  def rq_current_pos_mm(gripper_socket=1):
      pos_gripper = rq_current_pos(gripper_socket)
      pos_mm = gripper_to_mm(pos_gripper, gripper_socket)
      return round_value_2_dec(pos_mm)
  end

  def rq_current_pos_inches(gripper_socket=1):
      pos_gripper = rq_current_pos(gripper_socket)
      pos_mm = gripper_to_mm(pos_gripper, gripper_socket)
      pos_in = pos_mm / 25.4
      return round_value_2_dec(pos_in)
  end

  def rq_move_mm(pos_mm, gripper_socket=1):
      pos_gripper = mm_to_gripper(pos_mm, gripper_socket)
      rq_move(pos_gripper, gripper_socket)
  end

  def rq_move_and_wait_mm(pos_mm, gripper_socket=1):
      pos_gripper = mm_to_gripper(pos_mm, gripper_socket)
      rq_move_and_wait(pos_gripper, gripper_socket)
  end

  def rq_move_inches(pos_in, gripper_socket=1):
      pos_mm = pos_in * 25.4
      rq_move_mm(pos_mm, gripper_socket)
  end

  def rq_move_and_wait_inches(pos_in, gripper_socket=1):
      pos_mm = pos_in * 25.4
      rq_move_and_wait_mm(pos_mm, gripper_socket)
  end

  def get_closed_norm(gripper_socket):
      return gripper_closed_norm[gripper_socket - 1]
  end

  def get_open_norm(gripper_socket):
      return gripper_open_norm[gripper_socket - 1]
  end

  def get_closed_mm(gripper_socket):
      return gripper_closed_mm[gripper_socket - 1]
  end

  def get_open_mm(gripper_socket):
      return gripper_open_mm[gripper_socket - 1]
  end

  def set_closed_norm(closed_norm, gripper_socket):
      gripper_closed_norm[gripper_socket - 1] = closed_norm
  end

  def set_open_norm(open_norm, gripper_socket):
      gripper_open_norm[gripper_socket - 1] = open_norm
  end

  def set_closed_mm(closed_mm, gripper_socket):
      gripper_closed_mm[gripper_socket - 1] = closed_mm
  end

  def set_open_mm(open_mm, gripper_socket):
      gripper_open_mm[gripper_socket - 1] = open_mm
  end

  def gripper_to_mm(value_gripper, gripper_socket):
      closed_norm = get_closed_norm(gripper_socket)
      open_norm = get_open_norm(gripper_socket)
      closed_mm = get_closed_mm(gripper_socket)
      open_mm = get_open_mm(gripper_socket)

      value_norm = (value_gripper / 255) * 100

      slope = (closed_mm - open_mm) / (closed_norm - open_norm)
      value_mm = slope * (value_norm - closed_norm) + closed_mm

      if (value_mm > open_mm):
          value_mm_limited = open_mm
      elif (value_mm < closed_mm):
          value_mm_limited = closed_mm
      else:
          value_mm_limited = value_mm
      end

      return value_mm_limited
  end

  def mm_to_gripper(value_mm, gripper_socket):
      closed_norm = get_closed_norm(gripper_socket)
      open_norm = get_open_norm(gripper_socket)
      closed_mm = get_closed_mm(gripper_socket)
      open_mm = get_open_mm(gripper_socket)

      slope = (closed_norm - open_norm) / (closed_mm - open_mm)
      value_norm = (value_mm - closed_mm) * slope + closed_norm

      value_gripper = value_norm * 255 / 100

      if (value_gripper > 255):
          value_gripper_limited = 255
      elif (value_gripper < 0):
          value_gripper_limited = 0
      else:
          value_gripper_limited = round_value(value_gripper)
      end

      return value_gripper_limited
  end

  def round_value(value):
      value_mod = value % 1

      if(value_mod < 0.5):
          return floor(value)
      else:
          return ceil(value)
      end
  end

  def round_value_2_dec(value):
      value_x_100 = value * 100
      value_x_100_rounded = round_value(value_x_100)
      return value_x_100_rounded / 100
  end

  def clear_socket_buffer(gripper_socket="1", read_timeout = 0.1):
    byte_in_buffer = socket_read_byte_list(1, gripper_socket, read_timeout)

    while(byte_in_buffer[0] >= 1):
        byte_in_buffer = socket_read_byte_list(1, gripper_socket, read_timeout)
    end
  end

  def rq_set_gripper_socket_acquire_option(enabled=False):
      gripper_socket_acquire_option = enabled

      if(not enabled):
          gripper_1_socket_acquired = False
          gripper_2_socket_acquired = False
          gripper_3_socket_acquired = False
          gripper_4_socket_acquired = False
      end
  end

  def rq_acquire_gripper_socket(gripper_socket="1"):
      if(gripper_socket_acquire_option):
          rq_wait_gripper_socket_released(gripper_socket)
          enter_critical
              rq_set_gripper_socket_acquired(gripper_socket, True)
          exit_critical

          clear_socket_buffer(gripper_socket, 0.002)

          sync()
      end
  end

  def rq_release_gripper_socket(gripper_socket="1"):
      if(gripper_socket_acquire_option):
          rq_set_gripper_socket_acquired(gripper_socket, False)

          sync()
      end
  end

  def rq_set_gripper_socket_acquired(gripper_socket="1", acquired=False):
      if(gripper_socket == "1"):
          gripper_1_socket_acquired = acquired
      elif(gripper_socket == "2"):
          gripper_2_socket_acquired = acquired
      elif(gripper_socket == "3"):
          gripper_3_socket_acquired = acquired
      elif(gripper_socket == "4"):
          gripper_4_socket_acquired = acquired
      end
  end

  def rq_get_gripper_socket_acquired(gripper_socket="1"):
      if(gripper_socket == "1"):
          return gripper_1_socket_acquired
      elif(gripper_socket == "2"):
          return gripper_2_socket_acquired
      elif(gripper_socket == "3"):
          return gripper_3_socket_acquired
      elif(gripper_socket == "4"):
          return gripper_4_socket_acquired
      end

      sync()
  end

  def rq_wait_gripper_socket_released(gripper_socket="1"):
      while(rq_get_gripper_socket_acquired(gripper_socket)):
          sync()
      end

      sync()
  end

  def scale(value, rawRange, scaledRange):
      def computeSlope(inputRange, outputRange):
          outputRangeDelta = outputRange[1] - outputRange[0]
          inputRangeDelta = inputRange[1] - inputRange[0]

          if (inputRangeDelta == 0):
              return 0
          else:
              return outputRangeDelta / inputRangeDelta
          end
      end

      def computeIntercept(slope, inputRange, outputRange):
          return outputRange[0] - (slope * inputRange[0])
      end

      def clipScaledValue(outputScaledValue, outputRange):
          if (outputRange[0] < outputRange[1]):
              return clipWhenLowerLimitIsLessThanHigher(outputScaledValue, outputRange)
          else:
              return clipWhenLowerLimitIsGreaterThanHigherLimit(outputScaledValue, outputRange)
          end
      end

      def clipWhenLowerLimitIsGreaterThanHigherLimit(outputScaledValue, outputRange):
          if (outputScaledValue < outputRange[1]):
              return outputRange[1]
          elif (outputScaledValue > outputRange[0]):
              return outputRange[0]
          else:
              return outputScaledValue
          end
      end

      def clipWhenLowerLimitIsLessThanHigher(outputScaledValue, outputRange):
          if (outputScaledValue < outputRange[0]):
              return outputRange[0]
          elif (outputScaledValue > outputRange[1]):
              return outputRange[1]
          else:
              return outputScaledValue
          end
      end

      slope = computeSlope(rawRange, scaledRange)
      intercept = computeIntercept(slope, rawRange, scaledRange)
      scaledValue = slope * value + intercept
      return clipScaledValue(scaledValue, scaledRange)
  end

  def limit(value, range):
      return scale(value, range, range)
  end


  rq_obj_detect = 0
  rq_init_comm_if_connected(9, "1")
  rq_init_comm_if_connected(2, "2")
  rq_init_comm_if_connected(3, "3")
  rq_init_comm_if_connected(4, "4")
  rq_print_connected_grippers()
  connectivity_checked = [-1,-1,-1,-1]
  status_checked = [-1,-1,-1,-1]
  current_speed = [-1,-1,-1,-1]
  current_force = [-1,-1,-1,-1]
  set_closed_norm(100.0, 1)
  set_open_norm(0.0, 1)
  set_closed_mm(0.0, 1)
  set_open_mm(50.0, 1)
  set_closed_norm(100.0, 2)
  set_open_norm(0.0, 2)
  set_closed_mm(0.0, 2)
  set_open_mm(50.0, 2)
  set_closed_norm(100.0, 3)
  set_open_norm(0.0, 3)
  set_closed_mm(0.0, 3)
  set_open_mm(50.0, 3)
  set_closed_norm(100.0, 4)
  set_open_norm(0.0, 4)
  set_closed_mm(0.0, 4)
  set_open_mm(50.0, 4)
  # end: URCap Installation Node
  $ 1 "BeforeStart"
  $ 2 "var_1≔ False "
  global var_1=  False
  $ 3 "thread_flag≔ False "
  global thread_flag=  False
  $ 4 "var_10≔[0,0,0,0,0,0,0,0,0,0]"
  global var_10=[0,0,0,0,0,0,0,0,0,0]
  $ 5 "Set"
  set_tcp(p[0.0,0.0,0.11,0.0,0.0,0.0])
  $ 198 "Thread_1"
  thread Thread_1():
    while (True):
      $ 199 "Loop thread_flag== False "
      while (thread_flag==  False  ):
        $ 200 "var_12=0"
        var_12=0
        $ 201 "Wait: 0.01"
        sleep(0.01)
      end
      $ 202 "Wait: 0.001"
      sleep(0.001)
      $ 203 "var_11≔get_tcp_force()"
      global var_11=get_tcp_force()
      $ 204 "If var_11[axis]*var_11[axis]<var_2[11]*var_2[11]"
      if (var_11[axis]*var_11[axis]<var_2[11]*var_2[11]):
        $ 205 "var_12=0"
        var_12=0
      else:
        $ 206 "Else"
        $ 207 "var_12=var_12+1"
        var_12=var_12+1
        $ 208 "If var_12>0"
        if (var_12>0):
          $ 209 "thread_flag= False "
          thread_flag=  False
        end
      end
    end
  end
  threadId_Thread_1 = run Thread_1()
  while (True):
    $ 6 "Robot Program"
    $ 7 "Loop var_1==False"
    while (var_1==False):
      $ 8 "var_1≔socket_open('192.168.1.5',30010)"
      global var_1=socket_open("192.168.1.5",30010)
      $ 9 "Wait: 0.5"
      sleep(0.5)
    end
    $ 10 "Loop var_1== True "
    thread Thread_while_10():
      while (True):
        $ 11 "Wait: 0.001"
        sleep(0.001)
        $ 12 "var_2≔socket_read_ascii_float(12)"
        global var_2=socket_read_ascii_float(12)
        $ 13 "Loop var_2[0]≠12"
        while (var_2[0] != 12):
          $ 14 "var_2≔socket_read_ascii_float(12)"
          global var_2=socket_read_ascii_float(12)
        end
        $ 15 "Switch var_2[1]"
        switch_1 = var_2[1]
        $ 16 "Case 0"
        if (0 == switch_1):
          $ 17 "'movejl'"
          # 'movejl'
          $ 18 "var_3≔p[var_2[2],var_2[3],var_2[4],var_2[5],var_2[6],var_2[7]]"
          global var_3=p[var_2[2],var_2[3],var_2[4],var_2[5],var_2[6],var_2[7]]
          $ 19 "movej(var_3,var_2[8],var_2[9],var_2[10],var_2[11])"
          movej(var_3,var_2[8],var_2[9],var_2[10],var_2[11])
          $ 20 "If var_2[12]==0"
          if (var_2[12]==0):
            $ 21 "socket_send_string('completed_pose_move')"
            socket_send_string("completed_pose_move")
          end
        elif (1 == switch_1):
          $ 22 "Case 1"
          $ 23 "'movej'"
          # 'movej'
          $ 24 "var_6≔[var_2[2],var_2[3],var_2[4],var_2[5],var_2[6],var_2[7]]"
          global var_6=[var_2[2],var_2[3],var_2[4],var_2[5],var_2[6],var_2[7]]
          $ 25 "movej(var_6,var_2[8],var_2[9],var_2[10],var_2[11])"
          movej(var_6,var_2[8],var_2[9],var_2[10],var_2[11])
          $ 26 "If var_2[12]==0"
          if (var_2[12]==0):
            $ 27 "socket_send_string('completed_joint_move')"
            socket_send_string("completed_joint_move")
          end
        elif (2 == switch_1):
          $ 28 "Case 2"
          $ 29 "'movel'"
          # 'movel'
          $ 30 "var_3≔p[var_2[2],var_2[3],var_2[4],var_2[5],var_2[6],var_2[7]]"
          global var_3=p[var_2[2],var_2[3],var_2[4],var_2[5],var_2[6],var_2[7]]
          $ 31 "movel(var_3,var_2[8],var_2[9],var_2[10],var_2[11])"
          movel(var_3,var_2[8],var_2[9],var_2[10],var_2[11])
          $ 32 "If var_2[12]==0"
          if (var_2[12]==0):
            $ 33 "socket_send_string('completed_linear_move')"
            socket_send_string("completed_linear_move")
          end
        elif (3 == switch_1):
          $ 34 "Case 3"
          $ 35 "'move to var_3 relative to current pose'"
          # 'move to var_3 relative to current pose'
          $ 36 "var_3≔p[var_2[2],var_2[3],var_2[4],var_2[5],var_2[6],var_2[7]]"
          global var_3=p[var_2[2],var_2[3],var_2[4],var_2[5],var_2[6],var_2[7]]
          $ 37 "var_5≔get_actual_tcp_pose()"
          global var_5=get_actual_tcp_pose()
          $ 38 "movel(pose_trans(var_5,var_3),var_2[8],var_2[9],var_2[10],var_2[11])"
          movel(pose_trans(var_5,var_3),var_2[8],var_2[9],var_2[10],var_2[11])
          $ 39 "If var_2[12]==0"
          if (var_2[12]==0):
            $ 40 "socket_send_string('completed_relative_linear_move')"
            socket_send_string("completed_relative_linear_move")
          end
        elif (4 == switch_1):
          $ 41 "Case 4"
          $ 42 "'force move in single axis'"
          # 'force move in single axis'
          $ 43 "var_5≔get_actual_tcp_pose()"
          global var_5=get_actual_tcp_pose()
          $ 44 "If var_2[2]≠0"
          if (var_2[2] != 0):
            $ 45 "var_5[0]=var_5[0]+var_2[2]"
            var_5[0]=var_5[0]+var_2[2]
            $ 46 "axis≔0"
            global axis=0
          else:
            $ 47 "ElseIf var_2[3]≠0"
            if (var_2[3] != 0):
              $ 48 "var_5[1]=var_5[1]+var_2[3]"
              var_5[1]=var_5[1]+var_2[3]
              $ 49 "axis≔1"
              global axis=1
            else:
              $ 50 "ElseIf var_2[4]≠0"
              if (var_2[4] != 0):
                $ 51 "var_5[2]=var_5[2]+var_2[4]"
                var_5[2]=var_5[2]+var_2[4]
                $ 52 "axis≔2"
                global axis=2
              end
            end
          end
          $ 53 "thread_flag= True "
          thread_flag=  True
          $ 54 "Loop thread_flag== True "
          thread Thread_while_54():
            while (True):
              $ 55 "movel(var_5,var_2[8],var_2[9],0,0)"
              movel(var_5,var_2[8],var_2[9],0,0)
              $ 56 "Wait: 0.01"
              sleep(0.01)
              $ 57 "thread_flag= False "
              thread_flag=  False
            end
          end
          if (thread_flag==  True  ):
            global thread_handler_54=run Thread_while_54()
            while (thread_flag==  True  ):
              sync()
            end
            kill thread_handler_54
          end
          $ 58 "stopl(10)"
          stopl(10)
          $ 59 "If var_2[12]==0"
          if (var_2[12]==0):
            $ 60 "socket_send_string('completed_force_move')"
            socket_send_string("completed_force_move")
          end
        elif (5 == switch_1):
          $ 61 "Case 5"
          $ 62 "'servoj'"
          # 'servoj'
          $ 63 "var_3≔p[var_2[2],var_2[3],var_2[4],var_2[5],var_2[6],var_2[7]]"
          global var_3=p[var_2[2],var_2[3],var_2[4],var_2[5],var_2[6],var_2[7]]
          $ 64 "If var_2[12]==0"
          if (var_2[12]==0):
            $ 65 "stopl(0.5)"
            stopl(0.5)
          else:
            $ 66 "Else"
            $ 67 "var_14≔get_inverse_kin(var_3)"
            global var_14=get_inverse_kin(var_3)
            $ 68 "servoj(var_14,t=var_2[9],lookahead_time=var_2[10],gain=var_2[11])"
            servoj(var_14,t=var_2[9],lookahead_time=var_2[10],gain=var_2[11])
          end
          $ 69 "If var_2[12]==0"
          if (var_2[12]==0):
            $ 70 "socket_send_string('completed_servoj_move')"
            socket_send_string("completed_servoj_move")
          end
        elif (6 == switch_1):
          $ 71 "Case 6"
          $ 72 "'speedl'"
          # 'speedl'
          $ 73 "var_6≔[var_2[2],var_2[3],var_2[4],var_2[5],var_2[6],var_2[7]]"
          global var_6=[var_2[2],var_2[3],var_2[4],var_2[5],var_2[6],var_2[7]]
          $ 74 "If var_2[10]==0"
          if (var_2[10]==0):
            $ 75 "speedl(var_6,var_2[8])"
            speedl(var_6,var_2[8])
          else:
            $ 76 "Else"
            $ 77 "speedl(var_6,var_2[8],var_2[10])"
            speedl(var_6,var_2[8],var_2[10])
          end
          $ 78 "socket_send_string('completed_speedl')"
          socket_send_string("completed_speedl")
        elif (7 == switch_1):
          $ 79 "Case 7"
          $ 80 "'speedj'"
          # 'speedj'
          $ 81 "var_6≔[var_2[2],var_2[3],var_2[4],var_2[5],var_2[6],var_2[7]]"
          global var_6=[var_2[2],var_2[3],var_2[4],var_2[5],var_2[6],var_2[7]]
          $ 82 "If var_2[10]==0"
          if (var_2[10]==0):
            $ 83 "speedj(var_6,var_2[8])"
            speedj(var_6,var_2[8])
          else:
            $ 84 "Else"
            $ 85 "speedj(var_6,var_2[8],var_2[10])"
            speedj(var_6,var_2[8],var_2[10])
          end
          $ 86 "socket_send_string('completed_speedj')"
          socket_send_string("completed_speedj")
        elif (8 == switch_1):
          $ 87 "Case 8"
          $ 88 "'stopl'"
          # 'stopl'
          $ 89 "stopl(var_2[8])"
          stopl(var_2[8])
          $ 90 "socket_send_string('completed_stopl')"
          socket_send_string("completed_stopl")
        elif (9 == switch_1):
          $ 91 "Case 9"
          $ 92 "'servoc'"
          # 'servoc'
          $ 93 "var_3≔p[var_2[2],var_2[3],var_2[4],var_2[5],var_2[6],var_2[7]]"
          global var_3=p[var_2[2],var_2[3],var_2[4],var_2[5],var_2[6],var_2[7]]
          $ 94 "If var_2[12]==0"
          if (var_2[12]==0):
            $ 95 "stopl(var_2[8])"
            stopl(var_2[8])
          else:
            $ 96 "Else"
            $ 97 "servoc(var_3,a=var_2[8],v=var_2[9],r=var_2[11])"
            servoc(var_3,a=var_2[8],v=var_2[9],r=var_2[11])
          end
          $ 98 "If var_2[12]==0"
          if (var_2[12]==0):
            $ 99 "socket_send_string('completed_servoc_move')"
            socket_send_string("completed_servoc_move")
          end
        elif (10 == switch_1):
          $ 100 "Case 10"
          $ 101 "'return current pose'"
          # 'return current pose'
          $ 102 "var_5≔get_actual_tcp_pose()"
          global var_5=get_actual_tcp_pose()
          $ 103 "socket_send_string(var_5)"
          socket_send_string(var_5)
        elif (11 == switch_1):
          $ 104 "Case 11"
          $ 105 "'return current joints'"
          # 'return current joints'
          $ 106 "var_4≔get_actual_joint_positions()"
          global var_4=get_actual_joint_positions()
          $ 107 "socket_send_string(var_4)"
          socket_send_string(var_4)
        elif (12 == switch_1):
          $ 108 "Case 12"
          $ 109 "'return inverse kin of pose'"
          # 'return inverse kin of pose'
          $ 110 "var_3≔p[var_2[2],var_2[3],var_2[4],var_2[5],var_2[6],var_2[7]]"
          global var_3=p[var_2[2],var_2[3],var_2[4],var_2[5],var_2[6],var_2[7]]
          $ 111 "socket_send_string(get_inverse_kin(var_3))"
          socket_send_string(get_inverse_kin(var_3))
        elif (13 == switch_1):
          $ 112 "Case 13"
          $ 113 "'return translation to get to 2nd pose from 1st pose coord system'"
          # 'return translation to get to 2nd pose from 1st pose coord system'
          $ 114 "var_3≔p[var_2[2],var_2[3],var_2[4],var_2[5],var_2[6],var_2[7]]"
          global var_3=p[var_2[2],var_2[3],var_2[4],var_2[5],var_2[6],var_2[7]]
          $ 115 "var_5≔get_actual_tcp_pose()"
          global var_5=get_actual_tcp_pose()
          $ 116 "socket_send_string(pose_trans(var_5,var_3))"
          socket_send_string(pose_trans(var_5,var_3))
        elif (14 == switch_1):
          $ 117 "Case 14"
          $ 118 "'return current forces'"
          # 'return current forces'
          $ 119 "socket_send_string(get_tcp_force())"
          socket_send_string(get_tcp_force())
        elif (15 == switch_1):
          $ 120 "Case 15"
          $ 121 "'return force magnitude'"
          # 'return force magnitude'
          $ 122 "socket_send_string(force())"
          socket_send_string(force())
        elif (16 == switch_1):
          $ 123 "Case 16"
          $ 124 "'return tool velocity'"
          # 'return tool velocity'
          $ 125 "socket_send_string(get_actual_tcp_speed())"
          socket_send_string(get_actual_tcp_speed())
        elif (17 == switch_1):
          $ 126 "Case 17"
          $ 127 "'return force magnitude'"
          # 'return force magnitude'
          $ 128 "socket_send_string(get_actual_joint_speeds())"
          socket_send_string(get_actual_joint_speeds())
        elif (20 == switch_1):
          $ 129 "Case 20"
          $ 130 "'set tcp'"
          # 'set tcp'
          $ 131 "var_3≔p[var_2[2],var_2[3],var_2[4],var_2[5],var_2[6],var_2[7]]"
          global var_3=p[var_2[2],var_2[3],var_2[4],var_2[5],var_2[6],var_2[7]]
          $ 132 "set_tcp(var_3)"
          set_tcp(var_3)
          $ 133 "If var_2[12]==0"
          if (var_2[12]==0):
            $ 134 "socket_send_string('tcp_updated')"
            socket_send_string("tcp_updated")
          end
        elif (21 == switch_1):
          $ 135 "Case 21"
          $ 136 "'set payload'"
          # 'set payload'
          $ 137 "set_payload(var_2[8],[var_2[2],var_2[3],var_2[4]])"
          set_payload(var_2[8],[var_2[2],var_2[3],var_2[4]])
          $ 138 "If var_2[12]==0"
          if (var_2[12]==0):
            $ 139 "socket_send_string('payload_updated')"
            socket_send_string("payload_updated")
          end
        elif (22 == switch_1):
          $ 140 "Case 22"
          $ 141 "'set digital out'"
          # 'set digital out'
          $ 142 "If var_2[9]==1"
          if (var_2[9]==1):
            $ 143 "set_configurable_digital_out(var_2[8], True )"
            set_configurable_digital_out(var_2[8],  True  )
          else:
            $ 144 "Else"
            $ 145 "set_configurable_digital_out(var_2[8], False )"
            set_configurable_digital_out(var_2[8],  False  )
          end
          $ 146 "If var_2[12]==0"
          if (var_2[12]==0):
            $ 147 "socket_send_string('digital output set')"
            socket_send_string("digital output set")
          end
        elif (30 == switch_1):
          $ 148 "Case 30"
          $ 149 "freedrive_mode()"
          freedrive_mode()
          $ 150 "socket_send_string('begin_freedrive_mode')"
          socket_send_string("begin_freedrive_mode")
        elif (31 == switch_1):
          $ 151 "Case 31"
          $ 152 "end_freedrive_mode()"
          end_freedrive_mode()
          $ 153 "socket_send_string('end_freedrive_mode')"
          socket_send_string("end_freedrive_mode")
        elif (32 == switch_1):
          $ 154 "Case 32"
          $ 155 "socket_send_string('begin_blend_move')"
          socket_send_string("begin_blend_move")
          $ 156 "var_13≔var_2[8]"
          global var_13=var_2[8]
          $ 157 "n≔0"
          global n=0
          $ 158 "Loop n<var_13"
          while (n<var_13):
            $ 159 "n=n+1"
            n=n+1
            $ 160 "Loop var_2[0]≠12"
            while (var_2[0] != 12):
              $ 161 "var_2≔socket_read_ascii_float(12)"
              global var_2=socket_read_ascii_float(12)
            end
            $ 162 "var_3≔p[var_2[2],var_2[3],var_2[4],var_2[5],var_2[6],var_2[7]]"
            global var_3=p[var_2[2],var_2[3],var_2[4],var_2[5],var_2[6],var_2[7]]
            $ 163 "var_10[n] = var_3"
            var_10[n] = var_3
          end
          $ 164 "movel(var_10[0],0.1,0.5,0,0)"
          movel(var_10[0],0.1,0.5,0,0)
          $ 165 "n≔0"
          global n=0
          $ 166 "Loop n<var_13"
          while (n<var_13):
            $ 167 "n=n+1"
            n=n+1
            $ 168 "movep(var_10[n])"
            movep(var_10[n])
          end
        elif (33 == switch_1):
          $ 169 "Case 33"
          $ 170 "socket_send_string('begin_blend_move')"
          socket_send_string("begin_blend_move")
        elif (40 == switch_1):
          $ 171 "Case 40"
          $ 172 "socket_send_string('robot_ready')"
          socket_send_string("robot_ready")
        elif (100 == switch_1):
          $ 173 "Case 100"
          $ 174 "'reset program'"
          # 'reset program'
          $ 175 "If var_2[12]==0"
          if (var_2[12]==0):
            $ 176 "socket_send_string('resetting...')"
            socket_send_string("resetting...")
          end
          $ 177 "socket_close()"
          socket_close()
          $ 178 "var_1≔ False "
          global var_1=  False
        elif (101 == switch_1):
          $ 179 "Case 101"
          $ 180 "socket_send_string('ready')"
          socket_send_string("ready")
        elif (400 == switch_1):
          $ 181 "Case 400"
          $ 182 "'safe move'"
          # 'safe move'
          $ 183 "var_3≔p[var_2[2],var_2[3],var_2[4],var_2[5],var_2[6],var_2[7]]"
          global var_3=p[var_2[2],var_2[3],var_2[4],var_2[5],var_2[6],var_2[7]]
          $ 184 "var_5≔get_actual_tcp_pose()"
          global var_5=get_actual_tcp_pose()
          $ 185 "var_7≔get_inverse_kin(var_3)"
          global var_7=get_inverse_kin(var_3)
          $ 186 "var_8≔get_inverse_kin(var_5)"
          global var_8=get_inverse_kin(var_5)
          $ 187 "var_9≔0"
          global var_9=0
          $ 188 "Loop 6 times"
          Loop_5 = 0
          while (Loop_5 < 6):
            $ 189 "If (var_7[Loop_5]-var_8[Loop_5])>2.0  or  (var_8[Loop_5]-var_7[Loop_5])>2.0"
            if ((var_7[Loop_5]-var_8[Loop_5])>2.0   or   (var_8[Loop_5]-var_7[Loop_5])>2.0):
              $ 190 "var_9=1"
              var_9=1
            end
            Loop_5 = Loop_5 + 1
          end
          $ 192 "If var_9==0"
          if (var_9==0):
            $ 193 "movej(var_3,1,var_2[8],0,0)"
            movej(var_3,1,var_2[8],0,0)
            $ 194 "socket_send_string('completed_pose_move')"
            socket_send_string("completed_pose_move")
          else:
            $ 195 "Else"
            $ 196 "socket_send_string('no_safe_move_found')"
            socket_send_string("no_safe_move_found")
          end
        end
      end
    end
    if (var_1==  True  ):
      global thread_handler_10=run Thread_while_10()
      while (var_1==  True  ):
        sync()
      end
      kill thread_handler_10
    end
  end
end
